FUNCTION_BLOCK AxisBase
VAR_INPUT
END_VAR
VAR_OUTPUT

END_VAR
VAR
	
	//bPower : BOOL;
	//bPowerStatus : BOOL;
	axis : AXIS_REF;
	fbPower : MC_Power;
	bEnablePositiveMovement AT %I* : BOOL := TRUE; //Feed enable in positive direction.
	bEnableNegativeMovement AT %I* : BOOL := TRUE; //Feed enable in negative direction.
	
	fbHome : MC_Home;
	

	
	AxisHomed : BOOL;
	
	//torque
	MaxTorque : LREAL;
	//MinTorque : LREAL;
	fbSoEread : FB_SoERead;
	
	//reset
	fbReset : MC_Reset;
	fBias: LREAL;
	fbSoeReset: FB_SoEReset;

	
	pActPosAdress : POINTER TO LREAL := 0;
END_VAR

axis.ReadStatus();

//bAxisError:=axis.Status.Error;
//bAxisDriveError:=axis.Status.DriveDeviceError;

AuxiliaryFunctions(axis);


	
fbPower(
	Axis:= axis, 
	Enable:= , 
	Enable_Positive:= bEnablePositiveMovement, 
	Enable_Negative:= bEnableNegativeMovement, 
	Override:= 100, 
	BufferMode:= ,
	Options:= , 
	Status=> , 
	Busy=> , 
	Active=> , 
	Error=> , 
	ErrorID=> );
	

fbHome(
	Axis:= axis, 
	Execute:= , 
	Position:= , 
	HomingMode:= MC_HomingMode.MC_Direct, 
	BufferMode:= , 
	Options:= , 
	bCalibrationCam:= , 
	Done=> , 
	Busy=> , 
	Active=> , 
	CommandAborted=> , 
	Error=> , 
	ErrorID=> );
	

fbSoEread(
Axis:= axis, 
NetId:= '', 
Idn:= S_0_IDNs + 82, 
Element:= 16#40, 
pDstBuf:= ADR(MaxTorque), 
BufLen:= SIZEOF(MaxTorque), 
Execute:= , 
Timeout:= , 
Busy=> , 
Error=> , 
AdsErrId=> , 
SercosErrId=> , 
Attribute=> );
	


IF fbSoeReset.Execute AND fbSoeReset.Busy THEN
	fbReset.Execute := FALSE;
END_IF

fbSOEReset(
	Axis:= axis , 
	NetId:= , 
	Execute:= , 
	Timeout:= , 
	Busy=> , 
	Error=> , 
	AdsErrId=> , 
	SercosErrId=> );
	

IF(pActPosAdress = 0) THEN
	pActPosAdress := ADR(axis.NcToPlc.ActPos);
END_IF

METHOD AuxiliaryFunctions : BOOL
VAR_INPUT
	axis : AXIS_REF;
END_VAR
VAR
	ReadMotorTemp  : BOOL;
	//fbBrakeControl : FB_BrakeControl;
	MotorTemperature: INT;
	Execute: INT;
	Timeout: INT;
	Busy: INT;
	fbReadMotorTemp: FB_SoEReadMotorTemperature;
	fbReadAmplifierTemp: FB_SoEReadAmplifierTemperature;
	
	fbClearEC : FB_EcMasterFrameStatisticClearTxRxErr;
	fbManualBrakeControlAX8000 : FB_CoEAX8000BrakeControl;
END_VAR

fbReadMotorTemp(
	Axis :=axis,
	NetId := ,
	Execute := ,
	Timeout := ,
	Busy => ,
	Error => ,
	AdsErrId => ,
	SercosErrId => ,
	MotorTemperature =>,
	Attribute => );
	
fbReadAmplifierTemp(
	Axis :=axis,
	NetId := ,
	Execute := ,
	Timeout := ,
	Busy => ,
	Error => ,
	AdsErrId => ,
	SercosErrId => ,
	AmplifierTemperature =>,
	Attribute => );
(*
IF ReadMotorTemp THEN
	
fbBrakeControl(

 fbBrakeControl( 
    Axis            := Axis,
    Execute         := TRUE,
    Timeout         := DEFAULT_ADS_TIMEOUT,
    MotorTemperature => MotorTemperature
 );
 IF NOT fbReadMotorTemp.Busy THEN
    fbReadMotorTemp(Axis := Axis, Execute := FALSE);
    ReadMotorTemp := FALSE;
 END_IF
END_IF 
*)
fbClearEC(sNetId := ,
	nEcMasterDevID := ,
	bExecute :=,
	tTimeout:=,
	bBusy =>,
	bError=>,
	nErrId=>);
	
fbManualBrakeControlAX8000(
	Axis := axis,
	Execute:=,
	Mode:=,
	Busy =>,
	Error=>,
	ErrorID=>);
END_METHOD

END_FUNCTION_BLOCK

(* stored: Version 1.1.0.1, ProductVersion 3.1.4024.12
   POU AxisBase: Id {3d7477b0-9d98-46c9-b003-cf67f4daff27}, SpecialFunc None
   Method AuxiliaryFunctions: Id {66dbbb86-a765-402b-94ea-bc3bf83ff02b} *)
